(*

.. <legal notes>

legal notes
=================
| SPDX-FileCopyrightText: © 2026 Oleksandr Tiutyk <trofimich@gmail.com>
| SPDX-License-Identifier: LGPL-3.0-only
| For details check: LGPL-3.0-only_

.. _LGPL-3.0-only: https://www.gnu.org/licenses/lgpl-3.0.en.html

.. </legal notes>

*)

INTERFACE IEmptyException EXTENDS IException

END_INTERFACE

(* stored: Version 1.1.0.1
   Itf IEmptyException: Id {17176714-5c64-47e1-941b-1bed8926f011} *)
